INTERFACE I_DeformationHandler

METHOD DeleteCachedCt : BOOL
VAR_INPUT
  iCT              : I_CT;
END_VAR
END_METHOD

END_INTERFACE

(* stored: Version 1.1.0.1, ProductVersion 3.1.4024.11
   Itf I_DeformationHandler: Id {d4a4c422-72f1-4982-9d32-cf63805782af}
   Method DeleteCachedCt: Id {cc6a910a-bc96-48d5-9448-7ead384a645b} *)
